fGEM1SetpointValue:= LIMIT(0,fGEM1SetpointValue,2);
if (NOT (GEM1_VVC_40.i_xExtILK_OK) OR (GEM1_VVC_40.M_IsClosed())) THEN
        eMode			:=eCTRL_MODE_PASSIVE;// eCTRL_MODE_RESET ;//eCTRL_MODE_PASSIVE;
        GEM1_VCN_40.M_ValveControl(CloseValve);
        fGEM1SetpointValue :=0;
 END_IF //Switch off the PID incase of interlock
if (GEM1_GO) THEN
    IF (bReset) THEN
        (* set the mode to RESET*)
        eMode							:= eCTRL_MODE_RESET   ;
        stCTRL_PID_PARAMS.fKp					:= fKp1;			(* proportional gain Kp				*)
        GEM1_VCN_40.M_ValveControl(CloseValve);
        //bReset := False;
    ELSE(* set the mode to ACTIVE --> normal operation *)
        fbCTRL_PID.bSync := FALSE;
        eMode							:= eCTRL_MODE_ACTIVE   ;
        GEM1_VCN_40.M_ValveControl(PressureControl);
    END_IF
END_IF

If(FTrig.Q)THEN
        eMode							:=eCTRL_MODE_PASSIVE;// eCTRL_MODE_RESET ;//eCTRL_MODE_PASSIVE;
        fbCTRL_PID.fManSyncValue :=0;
        fbCTRL_PID.bSync := TRUE;
        GEM1_VCN_40.M_ValveControl(CloseValve);
        fGEM1SetpointValue :=0;
END_IF


fbCTRL_LIN_INTERPOLATION(
    fIn:= fGEM1SetpointValue ,
    fManValue:= fManValue,
    bExtrapolate:= bExtrapolate,
    eMode:= eMode,
    fOut=> ,
    bInIsGreaterThanMaxElement=> ,
    bInIsLessThanMinElement=> ,
    eState=> ,
    eErrorId=> ,
    bError=> ,
    stParams:= stCTRL_LIN_INTERPOLATION_PARAMS_GEM );



(* call controller *)
fbCTRL_PID(		fSetpointValue		:= fGEM1SetpointValue,
                    fActualValue		:= ,
                    fManSyncValue	:= ,
                    bSync				:= bSync,
                    eMode				:= eMode,
                    bHold				:= bHold,
                    stParams			:= stCTRL_PID_PARAMS,
                    fOut				=>  ,
                    bARWactive		=> bARWactive,
                    eErrorId			=> eErrorId,
                    bError				=>
                );



(*deadband/clipper *)

(* call function block *)
stCTRL_DEADBAND_PARAMS.fThreshold	:=  fGEM1SetpointValue*0.0016 ;
(*fbCTRL_DEADBAND	(	fIn					:= ,
                    stParams			:= stCTRL_DEADBAND_PARAMS,
                    bInIsUnderThreshold => ,
                    eErrorId			=> ,
                    bError				=>
                );*)

bError := fbCTRL_PID.bError OR fbCTRL_LIN_INTERPOLATION.bError;


// or NOT???

//stCTRL_PID_PARAMS.bDInTheFeedbackPath := fbCTRL_DEADBAND.bInIsUnderThreshold;


//timer
//pid_on(IN:=, PT:= wait, Q=>, ET =>);
//IF (pid_on.Q) THEN eMode:= eCTRL_MODE_ACTIVE; pid_on.IN := FALSE; END_IF; //eCTRL_MODE_TUNE????

FTRIG(CLK := GEM1_GO);

END_PROGRAM

// ---- POUs/PRG_GEM2.TcPOU
PROGRAM PRG_GEM2
VAR
    {attribute 'pytmc' :='
     pv: EM2L0:GEM:CNTRL:RESET;
     field: ZNAM FALSE;
     field: ONAM TRUE;
     io: io;
    '}
    bReset : BOOL;
    {attribute 'pytmc' :=' pv: EM2L0:GEM:CNTRL:ERROR;
     field: ZNAM FALSE;
     field: ONAM TRUE;
     io: io;
     '}
    bError : BOOL;
    {attribute 'pytmc' :=' pv: EM2L0:GEM:CNTRL:Kp1 '}
    fKp1 : REAL:= 0.25;
    {attribute 'pytmc' :=' pv: EM2L0:GEM:CNTRL:Tn1 '}
    fTn1 : REAL:= 1;//0.5;
    {attribute 'pytmc' :=' pv: EM2L0:GEM:CNTRL:Kp2 '}
    fKp2 : REAL:= 0.01;
    {attribute 'pytmc' :=' pv: EM2L0:GEM:CNTRL:Tn2 '}
    fTn2 : REAL:= 0.5;
    arrTable_GEM2	: ARRAY[1..31,1..2] OF FLOAT;
    fManValue											: FLOAT;
    bExtrapolate										: BOOL;
    eMode							: E_CTRL_MODE;
    stCTRL_PID_PARAMS		: ST_CTRL_PID_PARAMS;
    bSync							: BOOL;
    bHold							: BOOL;
    eErrorId						: E_CTRL_ERRORCODES;
    bARWactive					: BOOL;
    (* controller *)
    fbCTRL_PID					: FB_CTRL_PID;
    bInit							: BOOL	:= TRUE;
    fbCTRL_LIN_INTERPOLATION					: FB_CTRL_LIN_INTERPOLATION;
    //stCTRL_LIN_INTERPOLATION_PARAMS		: ST_CTRL_LIN_INTERPOLATION_PARAMS;
    stCTRL_LIN_INTERPOLATION_PARAMS_GEM	: ST_CTRL_LIN_INTERPOLATION_PARAMS;
    fbCTRL_DEADBAND						: FB_CTRL_DEADBAND;
    stCTRL_DEADBAND_PARAMS			: ST_CTRL_DEADBAND_PARAMS;
        //timer to switch the pid from manual to active 5seconds??? 10 seconds???
    pid_on :TON;
    wait : time := T#10S;
    FTrig: F_TRIG;




END_VAR


(*Devices*)
(*Gauges*)
GEM2_GCM_41(i_rFULL_SCALE := 2.0 (*Torr*));
GEM2_GCM_42(i_rFULL_SCALE := 0.05 (*Torr*));
(*Assign reading to psuedo gauge*)
IF (GEM2_GCM_42.PG.rPRESS >0.04) THEN GEM2_GCM_40 := GEM2_GCM_41.PG;
    ELSE
    GEM2_GCM_40 := GEM2_GCM_42.PG;
END_IF
(* Gauge selection *)
    fbCTRL_PID.fActualValue := GEM2_GCM_40.rPRESS;
(*
IF (fGEM2SetpointValue >0.04) THEN
    fbCTRL_PID.fActualValue := GEM2_GCM_41.PG.rPRESS;
ELSE
    fbCTRL_PID.fActualValue := GEM2_GCM_42.PG.rPRESS;
END_IF*)
(* N2 Cut Off Valves *)
GEM2_VVC_40(i_xExtILK_OK:= GEM2_Aperture_Closed AND GEM2_Turbo_Valves_Open AND GEM2_Turbo_Running);
(*Flow Control Valves*)
GEM2_VCN_40 (i_xExtIlkOK := (GEM2_Aperture_Closed AND GEM2_Turbo_Valves_Open AND GEM2_Turbo_Running),// AND GEM2_VVC_40.M_IsOpen()),
            i_ReqPos:=  fbCTRL_LIN_INTERPOLATION.fOut + fbCTRL_PID.fOut);

(*Iniitialization*)
IF bInit
THEN
    (* init array with the interpolation points  *)
    (* 	fIn					 |		fOut		*)
    arrTable_GEM2[1,1] := 0;		arrTable_GEM2[1,2] := 38.7;
    arrTable_GEM2[2,1] := 0.0000412;		arrTable_GEM2[2,2] := 38.8;
    arrTable_GEM2[3,1] := 0.001282;		arrTable_GEM2[3,2] := 38.9;
    arrTable_GEM2[4,1] :=  0.002136;	    arrTable_GEM2[4,2] := 39;
    arrTable_GEM2[5,1] :=  0.005884;	    arrTable_GEM2[5,2] := 40;
    arrTable_GEM2[6,1] := 0.00907;		arrTable_GEM2[6,2] := 42;
    arrTable_GEM2[7,1] := 0.01183;		arrTable_GEM2[7,2] := 44;
    arrTable_GEM2[8,1] := 0.01799;	    arrTable_GEM2[8,2] := 46;
    arrTable_GEM2[9,1] := 0.0302;	    arrTable_GEM2[9,2] := 47;
    arrTable_GEM2[10,1] := 0.0417;		arrTable_GEM2[10,2] := 50;
    arrTable_GEM2[11,1] := 0.06635;		arrTable_GEM2[11,2] := 51;
    arrTable_GEM2[12,1] := 0.08118;		arrTable_GEM2[12,2] := 53;
    arrTable_GEM2[13,1] := 0.0998;		arrTable_GEM2[13,2] := 56;
    arrTable_GEM2[14,1] := 0.10644;		arrTable_GEM2[14,2] := 56.5;
    arrTable_GEM2[15,1] := 0.1359;		arrTable_GEM2[15,2] := 58;
    arrTable_GEM2[16,1] := 0.1929;		arrTable_GEM2[16,2] := 60;
    arrTable_GEM2[17,1] := 0.2922;		arrTable_GEM2[17,2] := 62;
    arrTable_GEM2[18,1] := 0.3428;	    arrTable_GEM2[18,2] := 64;
    arrTable_GEM2[19,1] :=  0.405;;	    arrTable_GEM2[19,2] :=66;
    arrTable_GEM2[20,1] := 0.481;		arrTable_GEM2[20,2] := 68;
    arrTable_GEM2[21,1] := 0.5542;		arrTable_GEM2[21,2] := 69;
    arrTable_GEM2[22,1] := 0.6333;	    arrTable_GEM2[22,2] := 70;
    arrTable_GEM2[23,1] := 0.7901;	    arrTable_GEM2[23,2] := 72;
    arrTable_GEM2[24,1] := 0.9307;		arrTable_GEM2[24,2] := 73.04;
    arrTable_GEM2[25,1] := 1.0448;		arrTable_GEM2[25,2] := 73.64;
    arrTable_GEM2[26,1] := 1.31919;;		arrTable_GEM2[26,2] := 74.45;
    arrTable_GEM2[27,1] :=  1.324;		arrTable_GEM2[27,2] :=74.46;
    arrTable_GEM2[28,1] := 1.71941;	arrTable_GEM2[28,2] := 75;
    arrTable_GEM2[29,1] :=  1.963194;		arrTable_GEM2[29,2] :=75.5;
    arrTable_GEM2[30,1] := 1.99999;	arrTable_GEM2[30,2] := 75.505;
    arrTable_GEM2[31,1] := 2;	arrTable_GEM2[31,2] := 75.55;
    (* init parameter struct *)
    stCTRL_LIN_INTERPOLATION_PARAMS_GEM.tCtrlCycleTime					:= T#10ms;
    stCTRL_LIN_INTERPOLATION_PARAMS_GEM.tTaskCycleTime					:= T#10ms;
    stCTRL_LIN_INTERPOLATION_PARAMS_GEM.nDataTable_NumberOfRows		:= INT_TO_UINT(31);

    (*FBCNTRL*)
    (* init parameter struct *)
    stCTRL_PID_PARAMS.tCtrlCycleTime		:= T#10ms;
    stCTRL_PID_PARAMS.tTaskCycleTime		:= T#10ms;
    stCTRL_PID_PARAMS.fKp					:= fKp1;			(* proportional gain Kp				*)
    stCTRL_PID_PARAMS.tTn					:= T#500ms;		(*  Tn									*)
    stCTRL_PID_PARAMS.tTv					:= T#200ms;	(*  Tv									*)
    stCTRL_PID_PARAMS.tTd					:= T#200ms;	(*  Td									*)
    stCTRL_PID_PARAMS.fOutMaxLimit			:=  7;			(* maximum output limit				*)
    stCTRL_PID_PARAMS.fOutMinLimit			:=  -100;			(* minimum output limit				*)

    (* set the mode to ACTIVE --> normal operation *)
    eMode							:= eCTRL_MODE_PASSIVE   ;
    (* reset the init flag *)
    bInit							:= FALSE;
END_IF
(* set the addresses *)
    stCTRL_LIN_INTERPOLATION_PARAMS_GEM.pDataTable_ADR			:= ADR(arrTable_GEM2);
    stCTRL_LIN_INTERPOLATION_PARAMS_GEM.nDataTable_SIZEOF		:= SIZEOF(arrTable_GEM2);

fGEM2SetpointValue:= LIMIT(0,fGEM2SetpointValue,2);
if (NOT (GEM2_VVC_40.i_xExtILK_OK) OR (GEM2_VVC_40.M_IsClosed())) THEN
         eMode	:= eCTRL_MODE_PASSIVE;
        GEM2_VCN_40.M_ValveControl(CloseValve);
        fGEM2SetpointValue :=0;
END_IF //Switch off the PID incase of interlock
if (GEM2_GO) THEN
    IF (bReset) THEN
    (* set the mode to RESET*)
    eMode							:= eCTRL_MODE_RESET   ;
    stCTRL_PID_PARAMS.fKp					:= fKp1;			(* proportional gain Kp				*)
    GEM2_VCN_40.M_ValveControl(CloseValve);
    //bReset := False;
    ELSE
        (* set the mode to ACTIVE --> normal operation *)
    eMode							:= eCTRL_MODE_ACTIVE   ;
     GEM2_VCN_40.M_ValveControl(PressureControl);
    END_IF
END_IF
If(FTrig.Q)THEN
        eMode							:= eCTRL_MODE_PASSIVE;
        GEM2_VCN_40.M_ValveControl(CloseValve);
        fGEM2SetpointValue :=0;
END_IF


fbCTRL_LIN_INTERPOLATION(
    fIn:= fGEM2SetpointValue ,
    fManValue:= fManValue ,
    bExtrapolate:= bExtrapolate,
    eMode:= eMode,
    stParams:= stCTRL_LIN_INTERPOLATION_PARAMS_GEM,
    fOut=> ,
    bInIsGreaterThanMaxElement=> ,
    bInIsLessThanMinElement=> ,
    eState=> ,
    eErrorId=> ,
    bError=> );



(* call controller *)
fbCTRL_PID(		fSetpointValue		:= fGEM2SetpointValue,
                    fActualValue		:= ,
                    fManSyncValue	:= ,
                    bSync				:= bSync,
                    eMode				:= eMode,
                    bHold				:= bHold,
                    stParams			:= stCTRL_PID_PARAMS,
                    fOut				=> ,
                    bARWactive		=> bARWactive,
                    eErrorId			=> eErrorId,
                    bError				=>
                );


(*deadband/clipper *)

(* call function block *)
stCTRL_DEADBAND_PARAMS.fThreshold	:=  fGEM2SetpointValue*0.0016 ;
(*fbCTRL_DEADBAND	(	fIn					:= ,
                    stParams			:= stCTRL_DEADBAND_PARAMS,
                    bInIsUnderThreshold => ,
                    eErrorId			=> ,
                    bError				=>
                );*)

bError := fbCTRL_PID.bError OR fbCTRL_LIN_INTERPOLATION.bError;




// or NOT???

//stCTRL_PID_PARAMS.bDInTheFeedbackPath := fbCTRL_DEADBAND.bInIsUnderThreshold;


//timer
(*pid_on(IN:=, PT:= wait, Q=>, ET =>);
IF (pid_on.Q) THEN eMode:= eCTRL_MODE_ACTIVE; pid_on.IN := FALSE; END_IF; //eCTRL_MODE_TUNE????*)


FTRIG(CLK := GEM2_GO);

END_PROGRAM

// ---- POUs/PRG_PMPS.TcPOU
PROGRAM PRG_PMPS
VAR
 fbArbiterIO : FB_SubSysToArbiter_IO;
 test : bool;
 ar1 : bool;
 ar2 : bool;
  ar3 : bool;
 nReqID:UDINT;
 nReqRM:UDINT;
 bRemove:bool;
END_VAR

(*Fast Fault instantiation*)
g_FastFaultOutput1.bAutoReset :=TRUE;
g_FastFaultOutput2.bAutoReset :=TRUE;
g_FastFaultOutput1.Execute();
g_FastFaultOutput2.Execute();


(* Arbiter Instantiation*)
(*Arbiter one responsible for the aperture valves*)
fbArbiterIO(Arbiter := GVL_ILK.g_fbArbiter, fbFFHWO := GVL_ILK.g_FastFaultOutput1);
GVL_ILK.g_fbArbiter2.ElevateRequest(GVL_ILK.g_fbArbiter);
GVL_ILK.g_fbArbiter3.ElevateRequest(GVL_ILK.g_fbArbiter);

GVL_ILK.g_fbArbiter.AddRequest(nReqID:= 90  , stReqBP:= PMPS_GVL.cstFullBeam, sDevName := 'plc-lfe-gem');
GVL_ILK.g_fbArbiter2.AddRequest(nReqID:= 91  , stReqBP:= PMPS_GVL.cstFullBeam, sDevName := 'plc-lfe-gem');
GVL_ILK.g_fbArbiter3.AddRequest(nReqID:= 92  , stReqBP:= PMPS_GVL.cstFullBeam, sDevName := 'plc-lfe-gem');


ar1:=GVL_ILK.g_fbArbiter.CheckRequestInPool(nReqID);
ar2:=GVL_ILK.g_fbArbiter2.CheckRequestInPool(nReqID);
ar3:=GVL_ILK.g_fbArbiter3.CheckRequestInPool(nReqID);
if (bRemove) THEN
    GVL_ILK.g_fbArbiter.RemoveRequest(nReqRM);
     GVL_ILK.g_fbArbiter2.RemoveRequest(nReqRM);
    GVL_ILK.g_fbArbiter3.RemoveRequest(nReqRM);
END_IF

END_PROGRAM

// ---- POUs/FB_PressureSensor_PX219.TcPOU
FUNCTION_BLOCK FB_PressureSensor_PX219
VAR_OUTPUT
    {attribute 'pytmc' := 'pv:'}
    Sensor : ST_PressureSensor;
END_VAR

VAR_INPUT
    rDefaultSP : REAL; (* Must assign a default value at instantiation*)
END_VAR

VAR
    v : REAL;
    AlarmTOF : TOF;


    (*IOs to be linked*)
    i_iPRESS_R AT %I* :INT; // input Pressure // Link to analog Input
END_VAR

// for Omega PX219-xxx, signal 0-5VDC, corresponding to 16383 max

(* Real-value calculation *)

  IF Sensor.iPRESS_R > 16383 THEN; //Px219 max signal 5VDC, equal to beckhoff AO input 16383
       Sensor.rPRESS := -1;
     Sensor.xPStateAlarm:= TRUE;
     ELSE
         V:= 5.0*INT_TO_REAL(Sensor.iPRESS_R)/16383;
         Sensor.rPRESS := LREAL_TO_REAL(V/5.0*Sensor.rFull_Scale); //FULL scale in Psi for pressure tranducer
  END_IF

 (* Validate setpoint *)
    IF (Sensor.rPressSP < Sensor.rMinPressSP OR Sensor.rPressSP > Sensor.rMaxPressSP) THEN;
        Sensor.rPressSP := rDefaultSP;
    END_IF

 (* Set alarm bit when pressure lower and equal to setpoint, delay off for 60s*)

  AlarmTOF (IN := Sensor.rPRESS <= Sensor.rPressSP, PT := T#60S, Q => Sensor.xPstateAlarm);



 (*Soft IO Mapping*)
  ACT_IO();

ACTION ACT_IO:
Sensor.iPRESS_R := i_iPRESS_R;
END_ACTION

END_FUNCTION_BLOCK

// ---- POUs/DIAGNOSTICS.TcPOU
PROGRAM DIAGNOSTICS
VAR
    //Change the PLC String Name to the actual PLC NAME
    sPLCName :STRING := 'PLC-LFE-GEM';
    //Link the sAMSNetID to the Etherat Master netID
    i_sAMSNetID AT %I*: AMSNETID;
    // DO NOT CHANGE
    sAMSNetID : STRING; //used for EPICS PV
    sLibVersion_LCLS_General : STRING;(* := stLibVersion_LCLS_General.sVersion*) ;
    fbEcatDiag:FB_EcatDiag;
    bAllSlaveStateGood : BOOL;
    bMasterStateGood :BOOL;
    iMasterState: WORD;
    sMasterState:STRING;
    nSlaveNumber : UINT;
    aiSlaveStates: ARRAY[1..256] OF BYTE;
    aEcSlaveInfo :  ARRAY[1..256] OF ST_EcDevice;
END_VAR

// Instaniating a call to the fbEcatDiag
fbEcatDiag(
    I_AMSNetId:=i_sAMSNetID ,
    i_xFirstPass:= _TaskInfo[1].FirstCycle,
    q_xAllSlaveStatesGood=> bAllSlaveStateGood ,
    q_anTermStates=> aiSlaveStates,
    q_xMasterStateGood=>bMasterStateGood ,
    q_nMasterState=> iMasterState,
    q_sMasterState=> sMasterState ,
    q_astEcConfSlaveInfo=> aEcSlaveInfo ,
    q_nSlaves=> nSlaveNumber);

END_PROGRAM

// ---- POUs/FB_MPA.TcPOU
FUNCTION_BLOCK FB_MPA
VAR_INPUT
    (*EPS Interlock Bits*)
    ibInsertOK: BOOL;
    ibRetractOK: BOOL;
    ibOverrideInterlock:BOOL; (*if true interlocks are ignored*)
    // Reset fault
    {attribute 'pytmc' := '
    pv: FF_Reset
    '}
    i_xReset: BOOL;
    i_sDevName : T_MaxString :=  'MPA'; // Device name for diagnostic
    i_nTransitionRootID: UDINT; //A unique transition Root ID that is equal to or greater than 1000
END_VAR
VAR_OUTPUT
    {attribute 'pytmc' := '
    pv:
    '}
    q_stAct 	:	ST_MPA;
    {attribute 'pytmc' := '
    pv: MPS_FAULT
    '}
    xMPS_OK:BOOL;
    {attribute 'pytmc' := '
    pv: MOT_DONE
    '}
    xDone:Bool; // Motion is Done
END_VAR
VAR_IN_OUT
    io_fbFFHWO    :    FB_HardwareFFOutput;
    fbArbiter: FB_Arbiter();
END_VAR
VAR
    // PMPS
    tBPTMtimeout:TON;
    bMoving : BOOL;
    bDone :BOOL;
    ibPMPS_OK:BOOL;
    bptm: BeamParameterTransitionManager;
    // PMPS
    fbFF    :    FB_FastFault :=(
        i_DevName := 'MPA',
        i_Desc := 'Fault occurs when the device is moving',
        i_TypeCode := 16#1010);
    (*Init*)
    xFirstPass	:	BOOL;
    fbFSInit		:	R_TRIG;

    (* Timeouts*)
    tTimeOutDuration: TIME:= T#5S;
    tInserttimeout: TON;
    tRetracttimeout:TON;

    (*IO*)
    i_xInsertedLS	AT%I*: BOOL;
    i_xRetractedLS	AT%I*: BOOL;
    q_xInsert_DO	AT%Q*: BOOL;
    q_xRetract_DO	AT%Q*: BOOL;


    // For logging
    fbLogger : FB_LogMessage := (eSubsystem:=E_SubSystem.MOTION);
    ePrevState : E_PositionState;
    tErrorPresent : R_TRIG;
    tAction : R_TRIG; // Primary action of this device (OPN_DO, etc.)
    tOverrideActivated : R_TRIG;
END_VAR


(*Initialize*)
fbFSInit( CLK := TRUE, Q => xFirstPass);
(*IO Mapping*)
ACT_IO();

IF xFirstPass THEN
    q_stAct.eState := E_PositionState.INVALID;
    q_stAct.bRetract_SW := FALSE;
    q_stAct.bInsert_SW := FALSE;
    fbFF.i_DevName := i_sDevName;
END_IF


(* Manage States*)
IF q_stAct.i_bInLS AND  q_stAct.i_bOutLS THEN
    q_stAct.eState:=E_PositionState.INVALID;
ELSIF NOT q_stAct.i_bInLS AND q_stAct.i_bOutLS THEN
    q_stAct.eState:=E_PositionState.RETRACTED;
ELSIF q_stAct.i_bInLS AND NOT q_stAct.i_bOutLS THEN
    q_stAct.eState:=E_PositionState.INSERTED;
ELSIF NOT q_stAct.i_bInLS AND NOT q_stAct.i_bOutLS THEN
    q_stAct.eState:=E_PositionState.MOVING;
ELSE
    q_stAct.eState:=E_PositionState.INVALID;
END_IF

(*Set the Done signal*)
xDone := (q_stAct.bRetract_SW AND q_stAct.eState=E_PositionState.RETRACTED) OR (q_stAct.eState=E_PositionState.INSERTED AND q_stAct.bInsert_SW);


(*MPS FAULT*)
(**)
xMPS_OK := i_xInsertedLS XOR i_xRetractedLS;//(q_stAct.eState=RETRACTED) OR (q_stAct.eState=INSERTED);


(*PMPS PERMISSION*)


(* Can't have bRetract_SW and  bInsert_SW both be true*)
(*If (q_stAct.bRetract_SW) and (q_stAct.bInsert_SW) THEN
    q_stAct.bRetract_SW := FALSE;
    q_stAct.bInsert_SW := FALSE;
END_IF*)

q_stAct.bRetractOK := ibRetractOK;
q_stAct.bInsertOK := ibInsertOK;

(*Actuate the device*)
q_stAct.q_bRetract := q_stAct.bRetractOK AND q_stAct.bRetract_SW;
q_stAct.q_bInsert := q_stAct.bInsertOK AND q_stAct.bInsert_SW;

IF q_stAct.q_bInsert THEN
    q_stAct.q_bRetract := FALSE;
    q_stAct.bRetract_SW:= FALSE;
ELSIF q_stAct.q_bRetract THEN
    q_stAct.q_bInsert := FALSE;
    q_stAct.bInsert_SW:= FALSE;
END_IF;


(*Timers*)
tInserttimeout(IN:= q_stAct.q_bInsert, PT := tTimeOutDuration );
tRetracttimeout(IN:= q_stAct.q_bRetract, PT := tTimeOutDuration);

///Check moving postion timout
IF NOT q_stAct.i_bInLS AND tInserttimeout.Q THEN
    q_stAct.bErrorPresent := TRUE;
ELSIF NOT q_stAct.i_bOutLS AND tRetracttimeout.Q THEN
    q_stAct.bErrorPresent := TRUE;
END_IF


(*FAST FAULT*)
fbFF(i_xOK := xMPS_OK,
    i_xReset := i_xReset,
    i_xAutoReset :=TRUE,
    io_fbFFHWO := io_fbFFHWO);


(*Soft IO Mapping*)
ACT_IO();
(*Logger*)
ACT_Logger();
//ACT_PMPS();

ACTION ACT_IO:
(*Inputs*)
q_stAct.i_bInLS :=  i_xInsertedLS;
q_stAct.i_bOutLS := i_xRetractedLS;

(*outputs*)
q_xInsert_DO:=q_stAct.q_bInsert;
q_xRetract_DO:=q_stAct.q_bRetract;
END_ACTION

ACTION ACT_Logger:


//Position STATE Logger
IF ePrevState <> q_stAct.eState THEN
      CASE q_stAct.eState OF
        E_PositionState.INVALID:
            fbLogger(sMsg:='Device is in invalid position.', eSevr:=TcEventSeverity.Critical);
          E_PositionState.MOVING:
            fbLogger(sMsg:='Device moving', eSevr:=TcEventSeverity.Warning);
        E_PositionState.RETRACTED:
            fbLogger(sMsg:='Device retracted.', eSevr:=TcEventSeverity.Info);
        E_PositionState.INSERTED:
            fbLogger(sMsg:='Device inserted.', eSevr:=TcEventSeverity.Info);
      END_CASE
      ePrevState := q_stAct.eState;
  END_IF



// Log valve open
tAction(CLK:= q_stAct.q_bRetract XOR q_stAct.q_bInsert);
IF tAction.Q THEN fbLogger(sMsg:='Device commanded to actuate', eSevr:=TcEventSeverity.Info); END_IF
END_ACTION

ACTION ACT_PMPS:
//bMoving := ((q_stAct.bRetract_SW OR NOT q_stAct.bInsert_SW) AND q_stAct.i_bInLS) XOR  ((NOT q_stAct.bRetract_SW OR q_stAct.bInsert_SW) AND q_stAct.i_bOutLS);
//bDone :=  ((q_stAct.bRetract_SW OR NOT q_stAct.bInsert_SW) AND q_stAct.i_bOutLS) XOR ((NOT q_stAct.bRetract_SW OR q_stAct.bInsert_SW) AND q_stAct.i_bInLS);

bptm(fbArbiter:=fbArbiter,
     i_TransitionAssertionID:=i_nTransitionRootID+2,
     i_stTransitionAssertion:=PMPS_GVL.cst0RateBeam,
     i_nRequestedAssertionID:=i_nTransitionRootID+ BOOL_TO_UDINT(q_stAct.bRetract_SW AND NOT q_stAct.bInsert_SW ),
     i_stRequestedAssertion:=,
     i_xMoving:=NOT xDone,
     i_xDoneMoving:= xDone,
     stCurrentBeamParameters:=PMPS_GVL.stCurrentBeamParameters,
     q_xTransitionAuthorized=>);

     // Timeout
tBPTMtimeout(IN:= bptm.i_xMoving AND NOT bptm.q_xTransitionAuthorized , PT:=T#1S);
ibPMPS_OK := bptm.q_xTransitionAuthorized OR tBPTMtimeout.Q;
END_ACTION

END_FUNCTION_BLOCK

// ---- POUs/FB_VGC_1.TcPOU
(* This function block implements basic functionality for Isolation Gate Valves*)
(* This function block interlock is as follows:
1. The valve can be opened when the difference between the pressures on both sides is
less than the maximum differential pressure.
2. This rule persists until the pressures on both sides are lower than the vacuum-setpoint.
3. Once at-vac, the valve will close if the pressure on either side rises above the setpoint.*)
(*This function block also implements PMPS and EPS interlocks, as well as Fast MPS trigger*)
{attribute 'no_check'}
{attribute 'reflection'}
FUNCTION_BLOCK FB_VGC_1 Extends FB_Valve
VAR_IN_OUT

END_VAR
VAR_INPUT
    (*Upstream Gauge, usually ion gauge*)
    i_stUSG	:	ST_VG;
    (*Downstream Gauge, usually ion gauge*)
    i_stDSG	:	ST_VG;
    {attribute 'pytmc' := '
    pv: Dis_DPIlk
    '}
    i_xDis_DPIlk : BOOL := FALSE;  (* Set to true when calling the function to disable the differential pressure interlock *)
    {attribute 'pytmc' := '
    pv: EPS_OK
    '}
    i_xEPS_OK:	BOOL	:= TRUE; (*External EPS interlock, Set to TRUE when no EPS interlock is required, otherwise set to correct interlock signal*)
    {attribute 'pytmc' := '
    pv: MPS_OK
    '}
    //i_xPMPS_OK:	BOOL	; (*External MPS interlock, Set to TRUE when no PMPS interlock is required*)
    i_xExt_OK: BOOL; (*Other External Interlock, Set to True when no external interlock is required. If this Valve is neigboring a Fast Shutter this should be linked to the fast shutter xVAC_FAULT_OK*)
    i_xOverrideMode : BOOL; (*To be linked to global override bit. This Overrides Vacuum logic only, EPS, MPS and PMPS are still enforces*)
    // Reset fault
    {attribute 'pytmc' := '
    pv: FF_Reset
    '}
    i_xReset: BOOL;
    i_xIsAperture:BOOL :=FALSE; // Set tp True if this is an Aperture Valve, the MPS Fault will trip only when moving.
    i_sDevName : T_MaxString :=  'VGC'; // Device name for diagnostic
    i_nTransitionRootID: UDINT; //A unique transition Root ID that is equalt to or greater than 1000
END_VAR
VAR_OUTPUT
    {attribute 'pytmc' := '
    pv:
    '}
    iq_stValve : ST_VGC; (* All valve data and states will be in this struct*)

    {attribute 'pytmc' := '
    pv: MPS_FAULT_OK
    field: ZNAM MPS FAULT ;
    field: ONAM MPS OK ;
    '}
    xMPS_OK:	BOOL; (*MPS Fast OK, is set when the Valve is Open*)
END_VAR
VAR_IN_OUT
    io_fbFFHWO    :    FB_HardwareFFOutput;
    fbArbiter: FB_Arbiter();
END_VAR
VAR
    // PMPS
    bMoving : BOOL;
    bDone :BOOL;
    i_xPMPS_OK:	BOOL;
    bptm: BeamParameterTransitionManager;
    FFO    :    FB_FastFault :=(
        i_DevName := 'VGC',
        i_Desc := 'Fault occurs when the valve is not in open state',
        i_TypeCode := 16#1010);
    //g_FastFaultOutput1	:	FB_HardwareFFOutput;

    {attribute 'instance-path'}
    {attribute 'noinit'}
    sPath: STRING;

    rDiffPressAllowed	:	REAL := 22.5; // Torr, Default value comes from Vat Valve Manual
    rDiffPress : REAL;
    set : BOOL;
    reset: BOOL;

    xFirstPass	:	BOOL;
    fbFSInit		:	R_TRIG;

    tonDelOK : TON;
    rtOK	:	R_TRIG;
    tonOvrd	:	TON;
    rtOpen	:	R_TRIG;
    ftClose: F_TRIG;

    tDelOK	:	TIME := T#60S;
    tOvrd	:	TIME := T#10s;


    (* Timeouts*)
    tTimeOutDuration: TIME:= T#30S;
    tOPNtimeout: TON;
    tCLStimeout:TON;
    tBPTMtimeout:TON;


    (*IO*)
    i_xOpnLS	AT%I*: BOOL;
    i_xClsLS	AT%I*: BOOL;
    q_xOPN_DO	AT%Q*: BOOL;

    // For logging
    eVGCPrevState : E_VGC;


END_VAR

(* Vacuum gate valve
A. Wallace
16-10-29

A gate valve isolates vacuum volumes. Ideally it can be opened when a system is vented
to allow for faster pumping, and will close when high vacuum is lost.

The following behavior is good for valves in something like a gas attenuator.
This function block does the following:
1. The valve can be opened when the difference between the pressures on both sides is
less than the maximum differential pressure.
2. This rule persists until the pressures on both sides are lower than the vacuum-setpoint.
3. Once at-vac, the valve will close if the pressure on either side rises above the setpoint.

Alternatively, the differential pressure interlock can be disabled so the valve may only be opened
if the pressure on both sides is lower than the at-vacuum-setpoint. You want this behavior if
the valve is to be used in a UHV section.

Hysteresis is employed to ensure a smooth transition from vented/pumping down, to at-vac.

Finally, an override system is built in so you can bypass all the interlocking logic and
get back online.
*)
(* 10/1/2018 Margaret Ghaly included EPS, PMPS Checkes and MPS trigger signals*)


fbFSInit( CLK := TRUE, Q => xFirstPass);
(*IO Mapping*)
ACT_IO();

(* On first PLC pass, put valve into vented state, which implies a closed valve *)
IF xFirstPass THEN
    iq_stValve.eVGC_State := Vented;
    iq_stValve.pv_xOPN_SW := FALSE;
    FFO.i_DevName := i_sDevName;
END_IF


///Check valve position
IF iq_stValve.i_xClsLS AND  iq_stValve.i_xOpnLS THEN
    iq_stValve.eState:=INVALID;
ELSIF NOT iq_stValve.i_xClsLS AND iq_stValve.i_xOpnLS AND iq_stValve.q_xOPN_DO THEN
    iq_stValve.eState:=OPEN;
ELSIF NOT iq_stValve.i_xClsLS AND iq_stValve.i_xOpnLS AND NOT iq_stValve.q_xOPN_DO THEN
    iq_stValve.eState:=OPEN_F;
ELSIF iq_stValve.i_xClsLS AND NOT iq_stValve.i_xOpnLS AND NOT iq_stValve.q_xOPN_DO THEN
    iq_stValve.eState:=CLOSED;
ELSIF NOT iq_stValve.i_xClsLS AND NOT iq_stValve.i_xOpnLS THEN
    iq_stValve.eState:=MOVING;
ELSE
    iq_stValve.eState:=INVALID;
END_IF

// Update hysteresis
///////////////////////////////////////////////////
IF iq_stValve.rAT_VAC_SP_LAST <> iq_stValve.rAT_VAC_SP OR xFirstPass THEN
    iq_stValve.rAT_VAC_SP_LAST := iq_stValve.rAT_VAC_SP;
    iq_stValve.rAT_VAC_HYS := iq_stValve.rHYST_PERC * iq_stValve.rAT_VAC_SP;
END_IF

iq_stValve.rAT_VAC_HYS := LIMIT(0, iq_stValve.rAT_VAC_HYS, iq_stValve.rAT_VAC_SP);
IF iq_stValve.rAT_VAC_SP <> 0 THEN
    IF iq_stValve.rHYST_PERC <> (iq_stValve.rAT_VAC_HYS / iq_stValve.rAT_VAC_SP) THEN
        iq_stValve.rHYST_PERC := LIMIT(0, (iq_stValve.rAT_VAC_HYS / iq_stValve.rAT_VAC_SP) ,1);
    END_IF
END_IF
// Valve at vacuum check
///////////////////////////////////////////////////
    set := i_stUSG.rPRESS < iq_stValve.rAT_VAC_HYS AND i_stDSG.rPRESS < iq_stValve.rAT_VAC_HYS AND i_stUSG.xPRESS_OK AND i_stDSG.xPRESS_OK;
     iq_stValve.xAT_VAC S= set;
    reset := i_stUSG.rPRESS > iq_stValve.rAT_VAC_SP OR i_stDSG.rPRESS > iq_stValve.rAT_VAC_SP OR NOT i_stUSG.xPRESS_OK OR NOT i_stDSG.xPRESS_OK;
    iq_stValve.xAT_VAC R= reset;

// Differential pressure check
///////////////////////////////////////////////////
    (* Calc the differential pressure across the valve *)
    rDiffPress := ABS(i_stUSG.rPRESS - i_stDSG.rPRESS);

    (* As long as the differential pressure is less than 30mbar, the valve is allowed to open *)
    IF rDiffPress <= rDiffPressAllowed AND i_stUSG.xPRESS_OK AND i_stDSG.xPRESS_OK THEN
        iq_stValve.xDP_OK := TRUE;
    ELSE
        iq_stValve.xDP_OK	:= FALSE;
        (* If the differential pressure is exceeded, even when the valve is open,
        the state is unexpected and triggers a fault, because it suggests that something
        is wrong with the valve, or gauges or mapping or there is a major leak on one side.*)
        iq_stValve.eVGC_State := ERR_DiffPress;
        iq_stValve.xERR_DifPres := TRUE;
    END_IF

// Valve state
///////////////////////////////////////////////////
CASE iq_stValve.eVGC_State OF
    Vented: (* The Vented state is used during pump down *)
        (* Assuming the pump down went well, we are now at vacuum on both sides,
        so we move to the vacuum state, otherwise remain in the vented state *)
        IF iq_stValve.xAT_VAC AND (NOT (iq_stValve.xERR_DifPres)) AND (NOT (iq_stValve.xERR_SP)) AND (NOT (iq_stValve.xERR_ExtFault))THEN
            iq_stValve.eVGC_State := AtVacuum;
        ELSE
            iq_stValve.eVGC_State := Vented;
        END_IF

    AtVacuum:
        IF iq_stValve.xAT_VAC THEN
        (* If both pressure setpoints are made,
        then enable the differential pressure interlock, regardless of the valve state
        assuming we're using some kind of ion gauge where a pressure setpoint cannot be higher than 1E-4 T *)
        iq_stValve.eVGC_State := AtVacuum;

        ELSE

            (* If the valve is open (or in an unknown state) and either gauge is not at it's vacuum setpoint,
            we have a loss of vacuum error *)
            IF (iq_stValve.i_xOpnLS OR (NOT iq_stValve.i_xOpnLS AND NOT iq_stValve.i_xClsLS)) THEN
                iq_stValve.eVGC_State := ERR_LostVac;
                iq_stValve.xERR_SP := TRUE; //TAW changed this to the ERR_SP bool because I think that's what it was intended to be?

            (* Alternatively, if the valve is already closed and we lose pressure on one side,
            it was probably intentional venting, so we calmly move back to venting mode, and
            disable the differential pressure interlock *) //??
            ELSIF iq_stValve.i_xClsLS THEN
                iq_stValve.eVGC_State := Vented;
            END_IF

        END_IF

    ERR_DiffPress:
        IF NOT (iq_stValve.xERR_DifPres) THEN
            IF iq_stValve.xAT_VAC AND (NOT (iq_stValve.xERR_DifPres)) AND (NOT (iq_stValve.xERR_SP)) AND (NOT (iq_stValve.xERR_ExtFault))THEN
                iq_stValve.eVGC_State := AtVacuum;
            ELSE
                iq_stValve.eVGC_State := Vented;
            END_IF
        END_IF


    ERR_LostVac:
        IF NOT (iq_stValve.xERR_SP) THEN
            IF iq_stValve.xAT_VAC AND (NOT (iq_stValve.xERR_DifPres)) AND (NOT (iq_stValve.xERR_SP)) AND (NOT (iq_stValve.xERR_ExtFault))THEN
                iq_stValve.eVGC_State := AtVacuum;
            ELSE
                iq_stValve.eVGC_State := Vented;
            END_IF
        END_IF

    ERR_ExtFault:
        IF NOT (iq_stValve.xERR_ExtFault) AND (i_xExt_OK) THEN
            IF iq_stValve.xAT_VAC AND (NOT (iq_stValve.xERR_DifPres)) AND (NOT (iq_stValve.xERR_SP)) AND (NOT (iq_stValve.xERR_ExtFault))THEN
                iq_stValve.eVGC_State := AtVacuum;
            ELSE
                iq_stValve.eVGC_State := Vented;
            END_IF
        END_IF
END_CASE

IF (NOT i_xExt_OK) AND (iq_stValve.eState=OPEN)  THEN
    iq_stValve.eVGC_State := ERR_ExtFault;
    iq_stValve.xERR_ExtFault := TRUE;
END_IF

// Interlock evaluation - with bypass for DP ILK bypass
///////////////////////////////////////////////
IF i_xDis_DPIlk THEN
    iq_stValve.xOPN_OK := iq_stValve.xEXT_OK; // AND iq_stValve.xDP_OK ;
ELSE
    iq_stValve.xOPN_OK := iq_stValve.xEXT_OK AND iq_stValve.xAT_VAC;
END_IF


(* Valve operation *)

(* Override logic *)
(* Goal: give ability to override, but do so in a way that people won't forget it.
Solution: Override only after ten seconds of override, protect against blips,
when the valve permission goes true for more than ten seconds consistently, remove override
*)

tonDelOK(IN:=iq_stValve.xOPN_OK, PT:=tDelOK);
rtOK(CLK:=tonDelOK.Q);
IF rtOK.Q AND iq_stValve.pv_xOvrdOpn THEN
    iq_stValve.pv_xOvrdOpn :=FALSE;
    if (iq_stValve.eState = OPEN) AND (i_xOverrideMode) THEN iq_stValve.pv_xOPN_SW := TRUE; END_IF //for seamless transition
    //Log
    fbLogger(sMsg:='Override expired', eSevr:=TcEventSeverity.Warning);
END_IF
// Release the Force Open bit when the system override is false
IF NOT (i_xOverrideMode) THEN  iq_stValve.pv_xOvrdOpn :=FALSE; END_IF
//Override timer
tonOvrd(IN:=iq_stValve.pv_xOvrdOpn, PT:=tOvrd);


(* Valve operation *)
(* Here's where we evaluate sw actions and operate the valve *)
(* Valve operation *)

ftClose(CLK:= iq_stValve.pv_xOPN_SW);
rtOpen(CLK:= iq_stValve.pv_xOPN_SW);
(*when interlock is lost the Valve closes regardless of the status of the PMPS and EPS*)
IF NOT (iq_stValve.xOPN_OK) THEN
    iq_stValve.pv_xOPN_SW:= FALSE; // Reset switch after inlk is lost
    iq_stValve.q_xOPN_DO := (iq_stValve.pv_xOPN_SW  AND iq_stValve.xOPN_OK) OR (tonOvrd.Q AND i_xOverrideMode);
ELSIF i_xPMPS_OK THEN
    iq_stValve.q_xOPN_DO := (iq_stValve.pv_xOPN_SW  AND iq_stValve.xOPN_OK) OR (tonOvrd.Q AND i_xOverrideMode);
//ELSIF NOT (i_xPMPS_OK) THEN
    // Only override mode
//	iq_stValve.q_xOPN_DO := (tonOvrd.Q AND i_xOverrideMode);
END_IF


(*MPS Fault setting*)
If (i_xIsAperture ) THEN
    (* When the valve  is open or in Closed position MPS is OK, Fault while moving*)
    xMPS_OK := i_xOpnLS XOR i_xClsLS;
ELSE
    (* When the valve  is open MPS is OK*)
    xMPS_OK := i_xOpnLS AND NOT i_xClsLS AND q_xOPN_DO;
END_IF


///Check valve moving postion timout
IF NOT iq_stValve.i_xClsLS AND tCLStimeout.Q THEN
    iq_stValve.bErrorPresent := TRUE;
    iq_stValve.sErrorMessage := 'Close Timeout';
ELSIF NOT iq_stValve.i_xOpnLS AND tOPNtimeout.Q THEN
    iq_stValve.bErrorPresent := TRUE;
    iq_stValve.sErrorMessage := 'Open Timeout';
END_IF
IF (iq_stValve.eState=INVALID) THEN
    iq_stValve.bErrorPresent := TRUE;
    iq_stValve.sErrorMessage := CONCAT(sPath,'Invalid Valve Position');
END_IF


(*Timers*)
tOPNtimeout(IN:= iq_stValve.q_xOPN_DO, PT := tTimeOutDuration );
tCLStimeout(IN:= NOT iq_stValve.q_xOPN_DO, PT := tTimeOutDuration);


// Alarm reset
//////////////////////////////////////
ACT_ResetAlarms();

(*IO Mapping*)
ACT_IO();

// Log States and triggers
ACT_Logger();

(*FAST FAULT*)
FFO(i_xOK := xMPS_OK,
    i_xReset := i_xReset,
    i_xAutoReset :=TRUE,
    io_fbFFHWO := io_fbFFHWO);

(*PMPS*)
ACT_PMPS();

ACTION ACT_IO:
(*inputs*)
iq_stValve.i_xOpnLS := 	i_xOpnLS;
iq_stValve.i_xClsLS:=	i_xClsLS;
iq_stValve.xEXT_OK := i_xEXT_OK;
iq_stValve.xOverrideMode := i_xOverrideMode;
(*outputs*)
q_xOPN_DO:= iq_stValve.q_xOPN_DO;

(*ILK Devices*)
iq_stValve.sIlkUSDeviceName := This^.i_stUSG.sPath;
iq_stValve.sIlkDSDeviceName := This^.i_stDSG.sPath;
END_ACTION

ACTION ACT_Logger:
// ILK logger

IF NOT (iq_stValve.xOPN_OK) AND (ePrevState = OPEN) AND NOT (TonOvrd.Q) THEN
         fbLogger(sMsg:='Lost interlock ok bit while valve was open.', eSevr:=TcEventSeverity.Critical);
END_IF


//Positiong STATE Logger
IF ePrevState <> iq_stValve.eState THEN
      CASE iq_stValve.eState OF
        INVALID:
            fbLogger(sMsg:='Valve invalid position.', eSevr:=TcEventSeverity.Critical);
          MOVING:
            fbLogger(sMsg:='Valve moving', eSevr:=TcEventSeverity.Warning);
        OPEN:
            fbLogger(sMsg:='Valve Open.', eSevr:=TcEventSeverity.Info);
        OPEN_F:
            fbLogger(sMsg:='Valve Open.', eSevr:=TcEventSeverity.Info);
        CLOSED:
            fbLogger(sMsg:='Valve closed.', eSevr:=TcEventSeverity.Info);
      END_CASE
      ePrevState := iq_stValve.eState;
  END_IF

 //Pressure STATE Logger
IF eVGCPrevState <> iq_stValve.eVGC_State THEN
      CASE iq_stValve.eVGC_State OF
        Vented:
             fbLogger(sMsg:='Vented', eSevr:=TcEventSeverity.Info);
          AtVacuum:
             fbLogger(sMsg:='Vacuum setpoint satisfied', eSevr:=TcEventSeverity.Info);
        ERR_DiffPress:
             fbLogger(sMsg:='Potential accidental vent.', eSevr:=TcEventSeverity.Critical);
        ERR_LostVac:
            fbLogger(sMsg:='Unexpected loss of vacuum while valve was open or moving.', eSevr:=TcEventSeverity.Critical);
        ERR_ExtFault:
             fbLogger(sMsg:='Lost external interlock while valve was open.', eSevr:=TcEventSeverity.Critical);
      END_CASE
      eVGCPrevState := iq_stValve.eVGC_State;
  END_IF



// Log valve timeouts
tErrorPresent(CLK:=iq_stValve.bErrorPresent);
IF tErrorPresent.Q THEN fbLogger(sMsg:=iq_stValve.sErrorMessage, eSevr:=TcEventSeverity.Warning); END_IF

// Log valve open
tAction(CLK:= iq_stValve.q_xOPN_DO);
IF tAction.Q THEN fbLogger(sMsg:='Valve commanded open', eSevr:=TcEventSeverity.Info); END_IF

// Log override mode enabled
tOverrideActivated(CLK:= (tonOvrd.Q AND i_xOverrideMode));
IF tOverrideActivated.Q THEN fbLogger(sMsg:='Valve override mode activated', eSevr:=TcEventSeverity.Warning); END_IF
END_ACTION

ACTION ACT_PMPS:
bMoving := (iq_stValve.pv_xOPN_SW AND iq_stValve.i_xClsLS) XOR (NOT iq_stValve.pv_xOPN_SW AND i_xOpnLS);
bDone := (iq_stValve.pv_xOPN_SW AND iq_stValve.i_xOpnLS) XOR (NOT iq_stValve.pv_xOPN_SW AND i_xClsLS);
If (i_xIsAperture ) OR (iq_stValve.pv_xOPN_SW )THEN
    bptm.i_stRequestedAssertion := PMPS_GVL.cstFullBeam;
ELSE  bptm.i_stRequestedAssertion := PMPS_GVL.cst0RateBeam;
END_IF
bptm(fbArbiter:=fbArbiter,
     i_TransitionAssertionID:=i_nTransitionRootID+2,
     i_stTransitionAssertion:=PMPS_GVL.cst0RateBeam,
     i_nRequestedAssertionID:=i_nTransitionRootID+ BOOL_TO_UDINT( iq_stValve.pv_xOPN_SW),
     i_stRequestedAssertion:=,
     i_xMoving:=bMoving,
     i_xDoneMoving:= bDone,
     stCurrentBeamParameters:=PMPS_GVL.stCurrentBeamParameters,
     q_xTransitionAuthorized=>);
// Timeout
tBPTMtimeout(IN:= bMoving AND NOT bptm.q_xTransitionAuthorized , PT:=T#1S);
i_xPMPS_OK := bptm.q_xTransitionAuthorized OR tBPTMtimeout.Q;
END_ACTION

ACTION ACT_ResetAlarms:
iq_stValve.xERR_DifPres R= iq_stValve.pv_xAlmRst;
iq_stValve.xERR_SP R= iq_stValve.pv_xAlmRst;
iq_stValve.bErrorPresent R= iq_stValve.pv_xAlmRst;
iq_stValve.xERR_ExtFault R= iq_stValve.pv_xAlmRst;

IF ( iq_stValve.pv_xAlmRst) THEN
    iq_stValve.sErrorMessage :='';
     iq_stValve.pv_xAlmRst := FALSE;
END_IF
END_ACTION

METHOD PUBLIC M_IsClosed : BOOL
VAR_INPUT
END_VAR
M_IsClosed := (This^.iq_stValve.eState = E_ValvePositionState.CLOSED);
END_METHOD

METHOD PUBLIC M_IsOpen : BOOL
VAR_INPUT
END_VAR
M_IsOpen := (This^.iq_stValve.eState = E_ValvePositionState.OPEN);
END_METHOD

// Use this Methode to Open or close the valve by setting the OPN_SW to the input value.
METHOD PUBLIC M_Set_OPN_SW : BOOL
VAR_INPUT
        value:BOOL;
END_VAR
This^.iq_stValve.pv_xOPN_SW := value;
END_METHOD

END_FUNCTION_BLOCK

// ---- POUs/PRG_SATT.TcPOU
PROGRAM PRG_SATT
VAR
    PMPS_OK: BOOL := TRUE; // to be linked to pmps
END_VAR

SATT_MPA_01(
    ibInsertOK:= PMPS_OK,
    ibRetractOK:= PMPS_OK ,
    //ibPMPS_OK:= PMPS_OK ,
    ibOverrideInterlock:= ,
    q_stAct=> ,
    xMPS_OK=> ,
    xDone=> ,
    i_xReset := ,
    io_fbFFHWO :=g_FastFaultOutput2,i_sDevName:= 'AT1L0:SOLID:MPA:01',fbArbiter:=g_fbArbiter3,
    i_nTransitionRootID:=5100);

SATT_MPA_02(
    ibInsertOK:= PMPS_OK,
    ibRetractOK:= PMPS_OK ,
    //ibPMPS_OK:= PMPS_OK ,
    ibOverrideInterlock:= ,
    q_stAct=> ,
    xMPS_OK=> ,
    xDone=> ,
    i_xReset := ,io_fbFFHWO :=g_FastFaultOutput2,i_sDevName:= 'AT1L0:SOLID:MPA:02',fbArbiter:=g_fbArbiter3,
    i_nTransitionRootID:=5200);

SATT_MPA_03(
    ibInsertOK:= PMPS_OK,
    ibRetractOK:= PMPS_OK ,
    //ibPMPS_OK:= PMPS_OK ,
    ibOverrideInterlock:= ,
    q_stAct=> ,
    xMPS_OK=> ,
    xDone=> ,
    i_xReset := ,io_fbFFHWO :=g_FastFaultOutput2,i_sDevName:= 'AT1L0:SOLID:MPA:03',fbArbiter:=g_fbArbiter3,
    i_nTransitionRootID:=5300);

SATT_MPA_04(
    ibInsertOK:= PMPS_OK,
    ibRetractOK:= PMPS_OK ,
    //ibPMPS_OK:= PMPS_OK ,
    ibOverrideInterlock:= ,
    q_stAct=> ,
    xMPS_OK=> ,
    xDone=> ,
    i_xReset := ,io_fbFFHWO :=g_FastFaultOutput2,i_sDevName:= 'AT1L0:SOLID:MPA:04',fbArbiter:=g_fbArbiter3,
    i_nTransitionRootID:=5400);

SATT_MPA_05(
    ibInsertOK:= PMPS_OK,
    ibRetractOK:= PMPS_OK ,
    //ibPMPS_OK:= PMPS_OK ,
    ibOverrideInterlock:= ,
    q_stAct=> ,
    xMPS_OK=> ,
    xDone=> ,
    i_xReset := ,io_fbFFHWO :=g_FastFaultOutput2,i_sDevName:= 'AT1L0:SOLID:MPA:05',fbArbiter:=g_fbArbiter3,
    i_nTransitionRootID:=5500);

SATT_MPA_06(
    ibInsertOK:= PMPS_OK,
    ibRetractOK:= PMPS_OK ,
    //ibPMPS_OK:= PMPS_OK ,
    ibOverrideInterlock:= ,
    q_stAct=> ,
    xMPS_OK=> ,
    xDone=> ,
    i_xReset := ,io_fbFFHWO :=g_FastFaultOutput2,i_sDevName:= 'AT1L0:SOLID:MPA:06',fbArbiter:=g_fbArbiter3,
    i_nTransitionRootID:=5600);

SATT_MPA_07(
    ibInsertOK:= PMPS_OK,
    ibRetractOK:= PMPS_OK ,
    //ibPMPS_OK:= PMPS_OK ,
    ibOverrideInterlock:= ,
    q_stAct=> ,
    xMPS_OK=> ,
    xDone=> ,
    i_xReset := ,io_fbFFHWO :=g_FastFaultOutput2,i_sDevName:= 'AT1L0:SOLID:MPA:07',fbArbiter:=g_fbArbiter3,
    i_nTransitionRootID:=5700);

SATT_MPA_08(
    ibInsertOK:= PMPS_OK,
    ibRetractOK:= PMPS_OK ,
    //ibPMPS_OK:= PMPS_OK ,
    ibOverrideInterlock:= ,
    q_stAct=> ,
    xMPS_OK=> ,
    xDone=> ,
    i_xReset := ,io_fbFFHWO :=g_FastFaultOutput2,i_sDevName:= 'AT1L0:SOLID:MPA:08',fbArbiter:=g_fbArbiter3,
    i_nTransitionRootID:=5800);

SATT_MPA_09(
    ibInsertOK:= PMPS_OK,
    ibRetractOK:= PMPS_OK ,
    //ibPMPS_OK:= PMPS_OK ,
    ibOverrideInterlock:= ,
    q_stAct=> ,
    xMPS_OK=> ,
    xDone=> ,
    i_xReset := ,io_fbFFHWO :=g_FastFaultOutput2,i_sDevName:= 'AT1L0:SOLID:MPA:09',fbArbiter:=g_fbArbiter3,
    i_nTransitionRootID:=5900);

(*
MPA_321();
MPA_322();
MPA_323();
MPA_324();
MPA_325();
MPA_326();
MPA_327();
MPA_328();
MPA_329(); *)

END_PROGRAM

// ---- POUs/PRG_SENSORS.TcPOU
PROGRAM PRG_SENSORS
VAR
        // Sensor Range in Psi
    CDA_SENS_PRESS_RANGE : REAL := 200;
    NITR_SENS_PRESS_RANGE: REAL := 200;
    H2O_SENS_PRESS_RANGE: REAL := 200;

    // Mim pressure setpoint in Psi
    CDA_SENS_MIN_PRESS_SP: REAL := 30;
    NITR_SENS_MIN_PRESS_SP: REAL := 15;
    H2O_SENS_MIN_PRESS_SP: REAL := 15;

    // Maximum pressure setpoint in Psi
    CDA_SENS_MAX_PRESS_SP: REAL := 160;
    NITR_SENS_MAX_PRESS_SP: REAL := 55;
    H2O_SENS_MAX_PRESS_SP: REAL := 80;

    // Press default setpoint in Psi
    CDA_SENS_DEFAULT_SP: REAL := 60;
    NITR_SENS_DEFAULT_SP: REAL := 25;
    H2O_SENS_DEFAULT_SP: REAL := 30;


END_VAR


GEM1_AIR_1(rDefaultSP:= CDA_SENS_DEFAULT_SP);
GEM1_AIR_2(rDefaultSP:= CDA_SENS_DEFAULT_SP);

GEM2_N2_1 (rDefaultSP:= NITR_SENS_DEFAULT_SP);
GEM2_N2_2 (rDefaultSP:= NITR_SENS_DEFAULT_SP);

END_PROGRAM
